{attribute 'GeneratedUsingTerminal: EL6851-0010-0016'}
{attribute addProperty BoxType "EL6851-0010-0016"}
{attribute addProperty Id "DMX_StatusAT %I*DMX_Status_5ECDEABE8DMX_Channel_1_64AT %I*DMX_Channel_005FDEFD64WcStateAT %I*WcState_9091E0EB2InfoDataAT %I*InfoData_94A18F5E2"}
{attribute addProperty CRC "2293335216"}
{attribute addProperty Size "76"}
TYPE EL6851_88B184B0 EXTENDS EtcSlaveTerminalBase_947E5A46 :
STRUCT
	{attribute addProperty Name "DMX_Status"}
	DMX_Status : DMX_Status_5ECDEABE;
	{attribute addProperty Name "DMX_Channel_1_64"}
	DMX_Channel_1_64 : DMX_Channel_005FDEFD;
	{attribute addProperty Name "WcState"}
	WcState : WcState_9091E0EB;
	{attribute addProperty Name "InfoData"}
	InfoData : InfoData_94A18F5E;
END_STRUCT
END_TYPE

(* stored: Version 1.2.0.0, ProductVersion 3.1.4024.9
   DUT EL6851_88B184B0: Id {74cd51d8-5d3a-4199-adcd-075484be4ca6} *)
